(* LS Electric XG5000 project: 241007_실습1자동물내림 *)
(* PLC LSPLC *)
(* module base 0 slot 0: 입력 모듈:XGI-D21A (DC 24V 입력, 8점 (전류소스/싱크입력)) *)
(* module base 0 slot 1: 출력 모듈:XGQ-RY1A (릴레이 출력, 8점 (2A용, 단독 COM.)) *)

PROGRAM NewProgram (* task: 스캔 프로그램 *)
VAR
    ON : TON;
    ON1 : TON;
    ON2 : TON;
    sec1 : TIME := T#1s;
    sec2 : TIME := T#2s;
    sec3 : TIME := T#3s;
    T0 : TON;
    T1 : TP;
    T2 : TP;
    time01 : TIME := T#1s; (* 1초 *)
    time02 : TIME := T#2s; (* 2초 *)
    time03 : TIME := T#3s; (* 3초 *)
    WATER : TP;
    WATER1 : TP;
    WATER2 : TOF;
    WATER3 : TOF;
    WATER4 : TP;
    WATER5 : TP;
    WATER6 : TOF;
    물1 AT %QX0.1.0 : BOOL;
    센서1 AT %IX0.0.0 : BOOL;
END_VAR

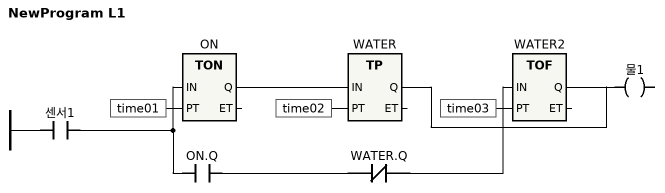
(* 사용자가 변기에 앉으면 1초 후, / 2초간 물이 나오고 / 이탈 후 즉시 3초간 물이 공급 *)
(* Rung L1 is block-masked: not executed *)
// ON(IN := 센서1, PT := time01);
// WATER(IN := ON.Q, PT := time02);
// WATER2(IN := 센서1 AND ON.Q AND NOT WATER.Q, PT := time03);
// 물1 := WATER.Q OR WATER2.Q;

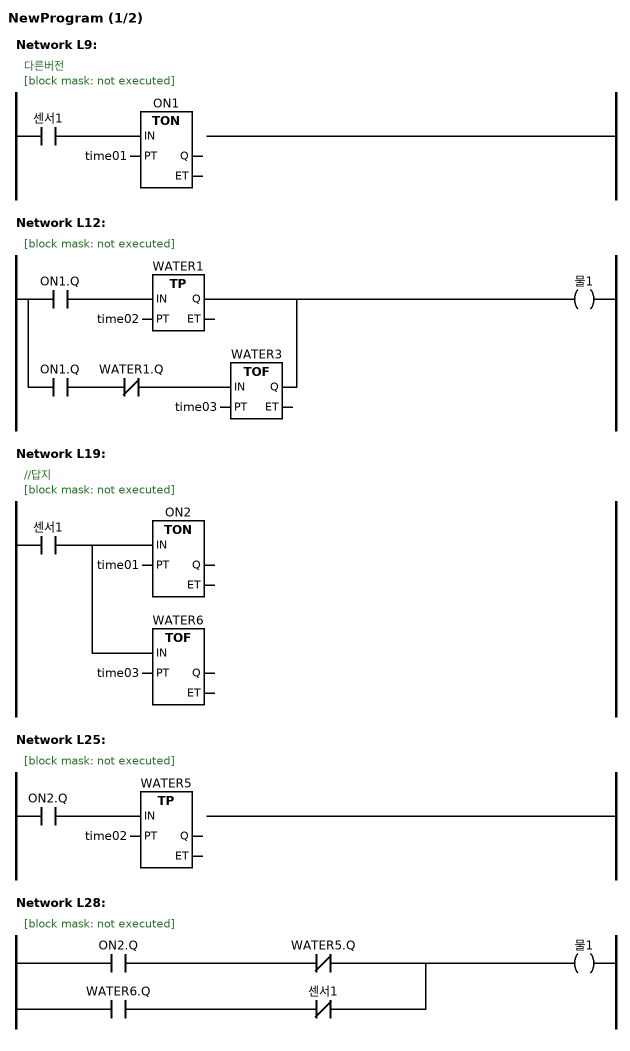
(* 다른버전 *)
(* Rung L9 is block-masked: not executed *)
// ON1(IN := 센서1, PT := time01);
(* Rung L12 is block-masked: not executed *)
// WATER1(IN := ON1.Q, PT := time02);
// WATER3(IN := ON1.Q AND NOT WATER1.Q, PT := time03);
// 물1 := WATER1.Q OR WATER3.Q;
(* //답지 *)
(* Rung L19 is block-masked: not executed *)
// ON2(IN := 센서1, PT := time01);
// WATER6(IN := 센서1, PT := time03);
(* Rung L25 is block-masked: not executed *)
// WATER5(IN := ON2.Q, PT := time02);
(* Rung L28 is block-masked: not executed *)
// 물1 := (ON2.Q AND NOT WATER5.Q) OR (WATER6.Q AND NOT 센서1);

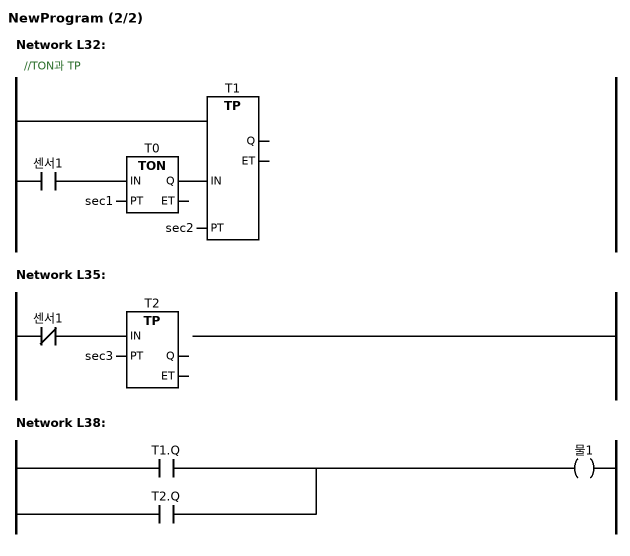
(* //TON과 TP *)
(* Rung L32 *)
T0(IN := 센서1, PT := sec1);
T1(IN := T0.Q, PT := sec2);
(* Rung L35 *)
T2(IN := NOT 센서1, PT := sec3);
(* Rung L38 *)
물1 := T1.Q OR T2.Q;
END_PROGRAM